ABB RAPID module: Module1.mod

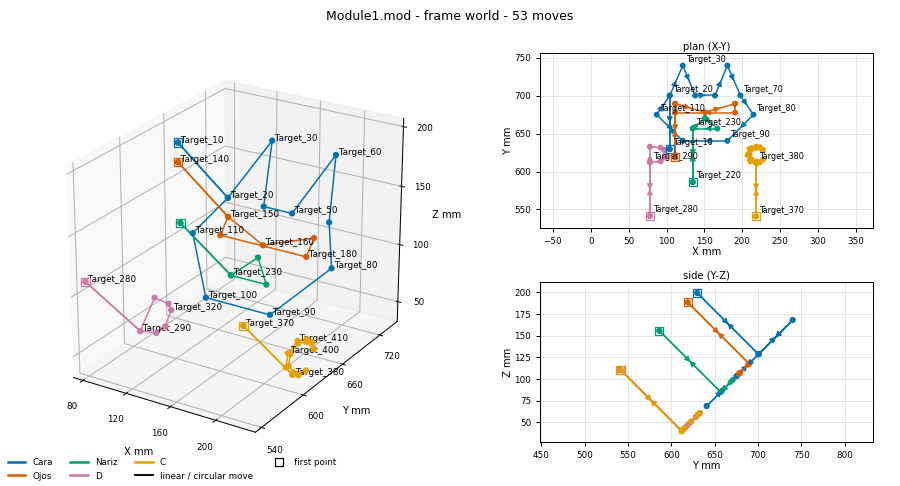
[picture p0: tool path of Module1.mod in frame world, 53 of 55 moves have a stored position in this frame; points joined in program order, loops and branches not executed]
MODULE Module1
        CONST robtarget Target_10:=[[-203.764162854,108.026112966,-100.000191688],[0.691676289,0,-0.000000001,0.722207665],[0,1,-2,0],[9E+09,9E+09,9E+09,9E+09,9E+09,9E+09]];
    CONST robtarget Target_20:=[[-203.764162854,108.026112862,-0.000191688],[0.691676289,0,-0.000000001,0.722207665],[0,1,-2,0],[9E+09,9E+09,9E+09,9E+09,9E+09,9E+09]];
    CONST robtarget Target_30:=[[-186.559461232,52.110827945,-0.000191746],[0.691676289,0,-0.000000001,0.722207665],[0,0,-2,0],[9E+09,9E+09,9E+09,9E+09,9E+09,9E+09]];
    CONST robtarget Target_40:=[[-170.191090842,108.026112855,-0.000191688],[0.691676289,0,-0.000000001,0.722207665],[0,1,-2,0],[9E+09,9E+09,9E+09,9E+09,9E+09,9E+09]];
    CONST robtarget Target_50:=[[-144.084389383,108.026112855,-0.000191688],[0.691676289,0,0,0.722207665],[0,1,-2,0],[9E+09,9E+09,9E+09,9E+09,9E+09,9E+09]];
    CONST robtarget Target_60:=[[-127.716018993,52.110827945,-0.000191746],[0.691676289,0.000000001,0,0.722207665],[0,0,-2,0],[9E+09,9E+09,9E+09,9E+09,9E+09,9E+09]];
    CONST robtarget Target_70:=[[-110.51131737,108.026112862,-0.000191688],[0.691676289,0.000000001,0,0.722207665],[0,1,-2,0],[9E+09,9E+09,9E+09,9E+09,9E+09,9E+09]];
    CONST robtarget Target_80:=[[-93.306615754,143.869244206,-0.00019165],[0.691676289,0.000000001,0,0.722207665],[0,1,-2,0],[9E+09,9E+09,9E+09,9E+09,9E+09,9E+09]];
    CONST robtarget Target_90:=[[-127.716018993,192.615902843,-0.000191599],[0.691676289,0,0,0.722207665],[0,1,-2,0],[9E+09,9E+09,9E+09,9E+09,9E+09,9E+09]];
    CONST robtarget Target_100:=[[-186.559461231,192.615902844,-0.000191599],[0.691676289,0,0,0.722207665],[0,1,-2,0],[9E+09,9E+09,9E+09,9E+09,9E+09,9E+09]];
    CONST robtarget Target_110:=[[-220.968864471,143.869244206,-0.00019165],[0.691676289,0,0,0.722207665],[0,1,-2,0],[9E+09,9E+09,9E+09,9E+09,9E+09,9E+09]];
    CONST robtarget Target_120:=[[-203.764162854,108.026112862,-0.000191688],[0.691676289,0,-0.000000001,0.722207665],[0,1,-2,0],[9E+09,9E+09,9E+09,9E+09,9E+09,9E+09]];
    CONST robtarget Target_130:=[[-203.764162854,108.026112966,-100.000191688],[0.691676289,0,-0.000000001,0.722207665],[0,1,-2,0],[9E+09,9E+09,9E+09,9E+09,9E+09,9E+09]];
    CONST robtarget Target_140:=[[-196.66181204,123.43497186,-100.000191672],[0.691676289,0.000000001,-0.000000001,0.722207665],[0,1,-2,0],[9E+09,9E+09,9E+09,9E+09,9E+09,9E+09]];
    CONST robtarget Target_150:=[[-196.66181204,123.434971754,-0.000191672],[0.691676289,0.000000001,-0.000000001,0.722207665],[0,1,-2,0],[9E+09,9E+09,9E+09,9E+09,9E+09,9E+09]];
    CONST robtarget Target_160:=[[-157.137740112,139.282664103,-0.000191655],[0.691676289,0.000000001,-0.000000001,0.722207665],[0,1,-2,0],[9E+09,9E+09,9E+09,9E+09,9E+09,9E+09]];
    CONST robtarget Target_170:=[[-117.613668185,123.434971754,-0.000191672],[0.691676289,0.000000001,-0.000000001,0.722207665],[0,1,-2,0],[9E+09,9E+09,9E+09,9E+09,9E+09,9E+09]];
    CONST robtarget Target_180:=[[-117.613668185,139.856817593,-0.000191654],[0.691676289,0,0,0.722207665],[0,1,-2,0],[9E+09,9E+09,9E+09,9E+09,9E+09,9E+09]];
    CONST robtarget Target_190:=[[-196.66181204,139.856817593,-0.000191654],[0.691676289,0,0,0.722207665],[0,1,-2,0],[9E+09,9E+09,9E+09,9E+09,9E+09,9E+09]];
    CONST robtarget Target_200:=[[-196.66181204,123.434971754,-0.000191672],[0.691676289,0,0,0.722207665],[0,1,-2,0],[9E+09,9E+09,9E+09,9E+09,9E+09,9E+09]];
    CONST robtarget Target_210:=[[-196.66181204,123.43497186,-100.000191672],[0.691676289,0,0,0.722207665],[0,1,-2,0],[9E+09,9E+09,9E+09,9E+09,9E+09,9E+09]];
    CONST robtarget Target_220:=[[-173.377942781,169.74257363,-100.000191623],[0.691676289,0,-0.000000001,0.722207665],[0,1,-2,0],[9E+09,9E+09,9E+09,9E+09,9E+09,9E+09]];
    CONST robtarget Target_230:=[[-173.377942781,169.742573525,-0.000191623],[0.691676289,0,-0.000000001,0.722207665],[0,1,-2,0],[9E+09,9E+09,9E+09,9E+09,9E+09,9E+09]];
    CONST robtarget Target_240:=[[-157.137740113,150.103708423,-0.000191643],[0.691676289,0,-0.000000001,0.722207665],[0,1,-2,0],[9E+09,9E+09,9E+09,9E+09,9E+09,9E+09]];
    CONST robtarget Target_250:=[[-140.897537443,169.742573525,-0.000191623],[0.691676289,0.000000001,0,0.722207665],[0,1,-2,0],[9E+09,9E+09,9E+09,9E+09,9E+09,9E+09]];
    CONST robtarget Target_260:=[[-173.377942781,169.742573525,-0.000191623],[0.691676289,0,0,0.722207665],[0,1,-2,0],[9E+09,9E+09,9E+09,9E+09,9E+09,9E+09]];
    CONST robtarget Target_270:=[[-173.377942781,169.74257363,-100.000191623],[0.691676289,0,0,0.722207665],[0,1,-2,0],[9E+09,9E+09,9E+09,9E+09,9E+09,9E+09]];
    CONST robtarget Target_280:=[[-229.97363672,233.029942704,-100.000191557],[0.691676289,0,0,0.722207665],[0,1,-2,0],[9E+09,9E+09,9E+09,9E+09,9E+09,9E+09]];
    CONST robtarget Target_290:=[[-229.97363672,233.0299426,-0.000191557],[0.691676289,0,0,0.722207665],[0,1,-2,0],[9E+09,9E+09,9E+09,9E+09,9E+09,9E+09]];
    CONST robtarget Target_300:=[[-229.97363672,203.690684295,-0.000191587],[0.691676289,0,0,0.722207665],[0,1,-2,0],[9E+09,9E+09,9E+09,9E+09,9E+09,9E+09]];
    CONST robtarget Target_310:=[[-215.883071876,205.427877221,-0.000191585],[0.691676289,0.000000001,-0.000000001,0.722207665],[0,1,-2,0],[9E+09,9E+09,9E+09,9E+09,9E+09,9E+09]];
    CONST robtarget Target_320:=[[-211.312600011,209.867370254,-0.000191581],[0.691676289,0,0,0.722207665],[0,1,-2,0],[9E+09,9E+09,9E+09,9E+09,9E+09,9E+09]];
    CONST robtarget Target_330:=[[-210.506046153,223.902786116,-0.000191567],[0.691676289,0,0,0.722207665],[0,1,-2,0],[9E+09,9E+09,9E+09,9E+09,9E+09,9E+09]];
    CONST robtarget Target_340:=[[-215.669369572,230.961855783,-0.000191558],[0.691676289,0,-0.000000001,0.722207665],[0,1,-2,0],[9E+09,9E+09,9E+09,9E+09,9E+09,9E+09]];
    CONST robtarget Target_350:=[[-229.97363672,233.0299426,-0.000191557],[0.691676289,0,0,0.722207665],[0,1,-2,0],[9E+09,9E+09,9E+09,9E+09,9E+09,9E+09]];
    CONST robtarget Target_360:=[[-229.97363672,233.029942704,-100.000191557],[0.691676289,0,0,0.722207665],[0,1,-2,0],[9E+09,9E+09,9E+09,9E+09,9E+09,9E+09]];
    CONST robtarget Target_370:=[[-89.840074026,233.609007014,-100.000191556],[0.691676289,0,0,0.722207665],[0,1,-2,0],[9E+09,9E+09,9E+09,9E+09,9E+09,9E+09]];
    CONST robtarget Target_380:=[[-89.840074026,233.609006909,-0.000191556],[0.691676289,0,0,0.722207665],[0,1,-2,0],[9E+09,9E+09,9E+09,9E+09,9E+09,9E+09]];
    CONST robtarget Target_390:=[[-97.464420757,229.431471539,-0.000191561],[0.691676289,0.000000001,-0.000000001,0.722207665],[0,1,-2,0],[9E+09,9E+09,9E+09,9E+09,9E+09,9E+09]];
    CONST robtarget Target_400:=[[-100.428678527,218.305164465,-0.000191572],[0.691676289,0,0,0.722207665],[0,1,-2,0],[9E+09,9E+09,9E+09,9E+09,9E+09,9E+09]];
    CONST robtarget Target_410:=[[-96.871569203,206.861750747,-0.000191584],[0.691676289,0,0,0.722207665],[0,1,-2,0],[9E+09,9E+09,9E+09,9E+09,9E+09,9E+09]];
    CONST robtarget Target_420:=[[-89.840074026,203.690684295,-0.000191587],[0.691676289,0,0,0.722207665],[0,1,-2,0],[9E+09,9E+09,9E+09,9E+09,9E+09,9E+09]];
    CONST robtarget Target_430:=[[-84.725005967,204.752302194,-0.000191587],[0.691676289,0,-0.000000001,0.722207665],[0,1,-2,0],[9E+09,9E+09,9E+09,9E+09,9E+09,9E+09]];
    CONST robtarget Target_440:=[[-81.429854306,209.770859536,-0.000191581],[0.691676289,0.000000001,-0.000000001,0.722207665],[0,1,-2,0],[9E+09,9E+09,9E+09,9E+09,9E+09,9E+09]];
    CONST robtarget Target_450:=[[-89.729776063,205.813920093,-0.000191585],[0.691676289,0,0,0.722207665],[0,1,-2,0],[9E+09,9E+09,9E+09,9E+09,9E+09,9E+09]];
    CONST robtarget Target_460:=[[-95.437695677,208.571369182,-0.000191583],[0.691676289,0,0,0.722207665],[0,1,-2,0],[9E+09,9E+09,9E+09,9E+09,9E+09,9E+09]];
    CONST robtarget Target_470:=[[-98.305442729,218.305164465,-0.000191572],[0.691676289,0,0,0.722207665],[0,1,-2,0],[9E+09,9E+09,9E+09,9E+09,9E+09,9E+09]];
    CONST robtarget Target_480:=[[-95.809951304,227.777002086,-0.000191562],[0.691676289,0.000000001,0,0.722207665],[0,1,-2,0],[9E+09,9E+09,9E+09,9E+09,9E+09,9E+09]];
    CONST robtarget Target_490:=[[-89.729776063,231.48577111,-0.000191559],[0.691676289,0,0,0.722207665],[0,1,-2,0],[9E+09,9E+09,9E+09,9E+09,9E+09,9E+09]];
    CONST robtarget Target_500:=[[-80.575045088,227.43232095,-0.000191562],[0.691676289,0.000000001,0,0.722207665],[0,1,-2,0],[9E+09,9E+09,9E+09,9E+09,9E+09,9E+09]];
    CONST robtarget Target_510:=[[-84.876665667,232.602537991,-0.000191557],[0.691676289,0.000000001,-0.000000001,0.722207665],[0,1,-2,0],[9E+09,9E+09,9E+09,9E+09,9E+09,9E+09]];
    CONST robtarget Target_520:=[[-89.840074026,233.609006909,-0.000191556],[0.691676289,0,0,0.722207665],[0,1,-2,0],[9E+09,9E+09,9E+09,9E+09,9E+09,9E+09]];
    CONST robtarget Target_530:=[[-89.840074026,233.609007014,-100.000191556],[0.691676289,0,0,0.722207665],[0,1,-2,0],[9E+09,9E+09,9E+09,9E+09,9E+09,9E+09]];
    CONST jointtarget h2:=[[0,0,0,0,0,0],[9E+09,9E+09,9E+09,9E+09,9E+09,9E+09]];
    CONST jointtarget H3:=[[0,30,0,0,50,0],[9E+09,9E+09,9E+09,9E+09,9E+09,9E+09]];
!***********************************************************
    !
    ! Module:  Module1
    !
    ! Description:
    !   <Insert description here>
    !
    ! Author: danny
    !
    ! Version: 1.0
    !
    !***********************************************************


    !***********************************************************
    !
    ! Procedure main
    !
    !   This is the entry point of your program
    !
    !***********************************************************
    PROC main()
        inicio;
        paso;
        Cara;
        Ojos;
        Nariz;
        D;
        C;
        paso;
        inicio;
    ENDPROC
    PROC Cara()
        MoveL Target_10,v150,z100,T_MakerHolder\WObj:=W_Board;
        MoveL Target_20,v150,z100,T_MakerHolder\WObj:=W_Board;
        MoveL Target_30,v150,z100,T_MakerHolder\WObj:=W_Board;
        MoveL Target_40,v150,z100,T_MakerHolder\WObj:=W_Board;
        MoveL Target_50,v150,z100,T_MakerHolder\WObj:=W_Board;
        MoveL Target_60,v150,z100,T_MakerHolder\WObj:=W_Board;
        MoveL Target_70,v150,z100,T_MakerHolder\WObj:=W_Board;
        MoveL Target_80,v150,z100,T_MakerHolder\WObj:=W_Board;
        MoveL Target_90,v150,z100,T_MakerHolder\WObj:=W_Board;
        MoveL Target_100,v150,z100,T_MakerHolder\WObj:=W_Board;
        MoveL Target_110,v150,z100,T_MakerHolder\WObj:=W_Board;
        MoveL Target_120,v150,z100,T_MakerHolder\WObj:=W_Board;
        MoveL Target_130,v150,z100,T_MakerHolder\WObj:=W_Board;
    ENDPROC
    PROC Ojos()
        MoveL Target_140,v150,z100,T_MakerHolder\WObj:=W_Board;
        MoveL Target_150,v150,z100,T_MakerHolder\WObj:=W_Board;
        MoveL Target_160,v150,z100,T_MakerHolder\WObj:=W_Board;
        MoveL Target_170,v150,z100,T_MakerHolder\WObj:=W_Board;
        MoveL Target_180,v150,z100,T_MakerHolder\WObj:=W_Board;
        MoveL Target_190,v150,z100,T_MakerHolder\WObj:=W_Board;
        MoveL Target_200,v150,z100,T_MakerHolder\WObj:=W_Board;
        MoveL Target_210,v150,z100,T_MakerHolder\WObj:=W_Board;
    ENDPROC
    PROC Nariz()
        MoveL Target_220,v150,z100,T_MakerHolder\WObj:=W_Board;
        MoveL Target_230,v150,z100,T_MakerHolder\WObj:=W_Board;
        MoveL Target_240,v150,z100,T_MakerHolder\WObj:=W_Board;
        MoveL Target_250,v150,z100,T_MakerHolder\WObj:=W_Board;
        MoveL Target_260,v150,z100,T_MakerHolder\WObj:=W_Board;
        MoveL Target_270,v150,z100,T_MakerHolder\WObj:=W_Board;
    ENDPROC
    PROC D()
        MoveL Target_280,v150,z100,T_MakerHolder\WObj:=W_Board;
        MoveL Target_290,v150,z100,T_MakerHolder\WObj:=W_Board;
        MoveL Target_300,v150,z100,T_MakerHolder\WObj:=W_Board;
        MoveL Target_310,v150,z100,T_MakerHolder\WObj:=W_Board;
        MoveL Target_320,v150,z100,T_MakerHolder\WObj:=W_Board;
        MoveL Target_330,v150,z100,T_MakerHolder\WObj:=W_Board;
        MoveL Target_340,v150,z100,T_MakerHolder\WObj:=W_Board;
        MoveL Target_350,v150,z100,T_MakerHolder\WObj:=W_Board;
        MoveL Target_360,v150,z100,T_MakerHolder\WObj:=W_Board;
    ENDPROC
    PROC C()
        MoveL Target_370,v150,z10,T_MakerHolder\WObj:=W_Board;
        MoveL Target_380,v150,z10,T_MakerHolder\WObj:=W_Board;
        MoveL Target_390,v150,z10,T_MakerHolder\WObj:=W_Board;
        MoveL Target_400,v150,z10,T_MakerHolder\WObj:=W_Board;
        MoveL Target_410,v150,z10,T_MakerHolder\WObj:=W_Board;
        MoveL Target_420,v150,z10,T_MakerHolder\WObj:=W_Board;
        MoveL Target_430,v150,z10,T_MakerHolder\WObj:=W_Board;
        MoveL Target_440,v150,z10,T_MakerHolder\WObj:=W_Board;
        MoveL Target_450,v150,z10,T_MakerHolder\WObj:=W_Board;
        MoveL Target_460,v150,z10,T_MakerHolder\WObj:=W_Board;
        MoveL Target_470,v150,z10,T_MakerHolder\WObj:=W_Board;
        MoveL Target_480,v150,z10,T_MakerHolder\WObj:=W_Board;
        MoveL Target_490,v150,z10,T_MakerHolder\WObj:=W_Board;
        MoveL Target_500,v150,z10,T_MakerHolder\WObj:=W_Board;
        MoveL Target_510,v150,z10,T_MakerHolder\WObj:=W_Board;
        MoveL Target_520,v150,z10,T_MakerHolder\WObj:=W_Board;
        MoveL Target_530,v150,z10,T_MakerHolder\WObj:=W_Board;
    ENDPROC
    PROC inicio()
        MoveAbsJ h2,v1000,z100,T_MakerHolder\WObj:=W_Board;
    ENDPROC
    PROC paso()
        MoveAbsJ H3,v1000,z100,T_MakerHolder\WObj:=W_Board;
    ENDPROC
ENDMODULE
